PROGRAM PRG_LD
VAR
END_VAR

// NETWORK 1

END_PROGRAM

(* stored: Version 1.1.0.1, ProductVersion 3.1.4024.12
   POU PRG_LD: Id {b87496fd-e94b-463e-acca-7889de6368b3}, SpecialFunc None *)
